// TIA Portal V16 export
// export: Created 2022-02-04T14:40:23.3972056Z, ExportSetting WithDefaults, DisplayName Totally Integrated Automation Portal, DisplayVersion V16 Update 1, DisplayName TIA Portal Version Control Interface, DisplayVersion V16, DisplayName TIA Portal Openness, DisplayVersion V16, DisplayName SINAMICS Startdrive Advanced, DisplayVersion V16 Update 5, DisplayName SINAMICS Startdrive G130, G150, S120, S150, SINAMICS MV, S210, DisplayVersion V16 Update 5, DisplayName SINAMICS Startdrive G110M, G120, G120C, G120D, G120P, G115D, DisplayVersion V16 Update 5, DisplayName STEP 7 Professional, DisplayVersion V16, DisplayName STEP 7 Safety, DisplayVersion V16, DisplayName WinCC Advanced, DisplayVersion V16, DisplayName SIMATIC Visualization Architect, DisplayVersion V16
DATA_BLOCK "SensLine_SigAdapter_DB"   // DB27
VERSION : 0.1
// stored: AutoNumber true, InstanceOfName SensLine_SigAdapter, InstanceOfType FB
"SensLine_SigAdapter"
   // VAR_INPUT
   //    InputSig : Word;
   // END_VAR
   // VAR_OUTPUT
   //    OutputSig : Word;
   // END_VAR
   // VAR RETAIN
   //    timer_18 : TON;
   //    timer_42 : TON;
   //    timer_48 : TON;
   //    timer_51 : TON;
   //    timer_57 { S7_SetPoint := 'True'} : TON;
   // END_VAR
BEGIN
END_DATA_BLOCK
